// TwinCAT 3 PLC project CL_DefectManagerPLC
// Title: CL_DefectManager
// Company: CleanGreens SA
// Author: Massimo Lucano
// ProjectVersion: 2.4
// Description: class to handle defects. Majour upgrade with several fixes and dynamic allocation
// ProgramVersion: 3.1.4024.0
// libraries:
//   CL_ErrorsDatabase, * (CleanGreens SA)
//   CL_CleanGreensObjectsLibrary, * (CleanGreens SA)
//   Tc2_Database, * (Beckhoff Automation GmbH)
//   Tc2_DataExchange, * (Beckhoff Automation GmbH)
//   Tc2_Standard, * (Beckhoff Automation GmbH)
//   Tc2_System, * (Beckhoff Automation GmbH)
//   Tc2_Utilities, * (Beckhoff Automation GmbH)
//   Tc3_Database, * (Beckhoff Automation GmbH)
//   Tc3_Module, * (Beckhoff Automation GmbH)
// project tree:
//   DUTs/ E_DefectState.TcDUT, ST_DefectManagerConstants.TcDUT, ST_DefectTable.TcDUT, T_DefectErrorID.TcDUT (not stored), T_InstancePath.TcDUT
//   GVLs/ CDefect.TcGVL
//   / PlcTask.TcTTO
//   POUs/ CL_Defect.TcPOU, CL_DefectManager.TcPOU, ITF_Defect.TcIO

CONFIGURATION CL_DefectManagerPLC
    RESOURCE PLC ON TwinCAT3
        TASK PlcTask(INTERVAL := T#10ms, PRIORITY := 20);
        PROGRAM MAIN WITH PlcTask : MAIN;
    END_RESOURCE
END_CONFIGURATION

// ---- DUTs/E_DefectState.TcDUT
{attribute 'qualified_only' := ''}
//{attribute 'strict'}   without strict type casting between integer et enum types is possible
TYPE E_DefectState :
(
	None := 0,
	Off,
	Active,
	ActiveAndAck,
	OffAndNotAck
);
END_TYPE

// ---- DUTs/ST_DefectManagerConstants.TcDUT
TYPE ST_DefectManagerConstants :
STRUCT
  nMaxDefects	        : UINT;//maximun number of defects that can be registred in the defect manager
	nMaxDefectsView	    :	UINT;//number of line to show in the HMI, each line is a defect
  nNumIrrLinesForHMI  : UINT;//number of irrigation line handled by a single PLC and HMI
END_STRUCT
END_TYPE

// ---- DUTs/ST_DefectTable.TcDUT
TYPE ST_DefectTable :
STRUCT
  bHideDefect   : BOOL := TRUE;
  pDefect       : pointer to CL_Defect; //pointer to the Defect itself
	State         : E_DefectState := E_DefectState.None;
	Severity      : TcEventSeverity := TcEventSeverity.Verbose;
	ErrorID       : STRING(3) :='';
	ClassID       : STRING(3) :='';
	Color         : DWORD := 0;
  InstancePath  : T_InstancePath := '';
	Description   : T_MaxString := '';
	RisingEdge    : STRING(CDefect.nDefectTableStrLen_C) := '';;
	FallingEdge   : STRING(CDefect.nDefectTableStrLen_C) := '';;
END_STRUCT
END_TYPE

// ---- DUTs/T_InstancePath.TcDUT
TYPE T_InstancePath : STRING(512); END_TYPE

// ---- GVLs/CDefect.TcGVL
{attribute 'qualified_only'}
VAR_GLOBAL CONSTANT
  //Defect manager library constants max array size
  nDefectTableStrLen_C        : UINT := 40;
	nMaxDefects_C    		        : UINT := 1000;
	nMaxDefectsView_C           : UINT := 40;
  tInfoOffTimeout_C           : TIME := T#5S; 
  tInfoOffAndNotAckTimeout_C  : TIME := T#15S;
END_VAR

// ---- POUs/ITF_Defect.TcIO
INTERFACE ITF_Defect EXTENDS __SYSTEM.IQueryInterface

METHOD Ack
END_METHOD

METHOD PUBLIC BuildStringMsg : BOOL
//return false if no error 
VAR_INPUT
	sMsgOut_P   : POINTER TO T_StringBuffer;//return the Telegram message
  sTextOut_P  : POINTER TO T_StringBuffer;//return the ADS console message  
  stShow      : ST_ShowMsgFields;
END_VAR
END_METHOD

PROPERTY PUBLIC CanSendAlarmMsg : BOOL
GET
END_GET
END_PROPERTY

PROPERTY PUBLIC CanSendInfoMsg : BOOL
GET
END_GET
END_PROPERTY

PROPERTY PUBLIC CanSendRegisterMsg : BOOL
GET
END_GET
END_PROPERTY

PROPERTY ClassID : STRING(3)
GET
END_GET
END_PROPERTY

METHOD PUBLIC DefectSentToFalse
VAR_INPUT
END_VAR
END_METHOD

PROPERTY PUBLIC Description : String
GET
END_GET
END_PROPERTY

PROPERTY ErrorID : STRING(3)
GET
END_GET
END_PROPERTY

PROPERTY FallingEdge : DATE_AND_TIME
GET
END_GET
END_PROPERTY

PROPERTY PUBLIC HideDefect : bool
GET
END_GET
END_PROPERTY

PROPERTY InstancePath : T_InstancePath
GET
END_GET
END_PROPERTY

METHOD PUBLIC Register : BOOL
VAR_INPUT
	DefectMngr  : REFERENCE TO CL_DefectManager;
  inClassID	  :	STRING(3);
  inErrorID   :	STRING(3);
END_VAR
END_METHOD

PROPERTY RisingEdge : DATE_AND_TIME
GET
END_GET
END_PROPERTY

METHOD PUBLIC Set
VAR_INPUT
  bSetActivate : BOOL;
END_VAR
END_METHOD

METHOD PUBLIC SetOff
VAR_INPUT
END_VAR
END_METHOD

METHOD PUBLIC SetOn
VAR_INPUT
END_VAR
END_METHOD

METHOD PUBLIC SetOnWithMsg
VAR_INPUT
  sAddMsg_P     : POINTER TO T_MaxString;
END_VAR
END_METHOD

METHOD PUBLIC SetWithMsg
VAR_INPUT
  bSetActivate  : BOOL;
  sAddMsg_P     : POINTER TO T_MaxString;
END_VAR
END_METHOD

PROPERTY Severity : TcEventSeverity
GET
END_GET
END_PROPERTY

PROPERTY State : E_DefectState
GET
END_GET
END_PROPERTY

METHOD UpdateHideDefect
END_METHOD

END_INTERFACE

// ---- POUs/CL_Defect.TcPOU
{attribute 'reflection'}
FUNCTION_BLOCK CL_Defect IMPLEMENTS ITF_Defect
VAR
 	_State              : E_DefectState := E_DefectState.None; 
	
	_ErrorIndex					:	UDINT;
	_ClassIndex					:	UDINT;
	
  _ErrorID            : STRING(3);
  _ClassID            : STRING(3);
  
	_DefectMngr	        : REFERENCE TO CL_DefectManager;
	_bRegistered		    : BOOL := FALSE;
	
	_Severity           : TcEventSeverity := TcEventSeverity.Critical;//temporary solution without database
		
	//used to send Telegram msg
	bTelAlarmSent       : BOOL := FALSE;
  bTelInfoSent        : BOOL := FALSE;
	bTelRegisteredSent	: BOOL := FALSE;
  
  bHideDefect	        : BOOL := true;
	
	_RisingEdge         : DATE_AND_TIME;
	_FallingEdge		    : DATE_AND_TIME;
	
	{attribute 'instance-path'}
	{attribute 'no_init'}
	_InstancePath       : T_InstancePath;
	InstanceStr_P		    : POINTER TO T_StringBuffer;
  _sAddMsg		        : string(64) := '';
END_VAR

METHOD PUBLIC Ack
IF State = E_DefectState.Active THEN
  _State := E_DefectState.ActiveAndAck;
ELSIF State = E_DefectState.OffAndNotAck THEN
  _State := E_DefectState.Off;
	DefectSentToFalse();
END_IF
END_METHOD

METHOD PUBLIC BuildStringMsg : BOOL
//return false if no error 
VAR_INPUT
	sMsgOut_P       : POINTER TO T_StringBuffer;//return the Telegram message
  sTextOut_P      : POINTER TO T_StringBuffer;//return the ADS console message  
  stShow          : ST_ShowMsgFields;
END_VAR
VAR
	bTmpErr			    : BOOL;
	bTmp1Err		    : BOOL;
  nErrIdOut       : UDINT;
	fbFormatStr	    : FB_FormatString;
  
	severityStr	    : T_MaxString;
	stateStr        : T_MaxString;
	sMsgAddLine	    :	T_MaxString;
  sMsgTmp         : T_MaxString;
  sClassID        : T_MaxString;
  sErrorID        : T_MaxString;
END_VAR
BuildStringMsg := FALSE;
sClassID := _ClassID;
sErrorID := _ErrorID;

CASE _State OF
		E_DefectState.None : stateStr := 'None';
		E_DefectState.Off : stateStr := 'Off';
		E_DefectState.Active : stateStr := 'Active';
		E_DefectState.ActiveAndAck : stateStr := 'ActiveAndAck';
		E_DefectState.OffAndNotAck : stateStr := 'OffAndNotAck';
END_CASE

CASE _Severity OF
		TcEventSeverity.Critical : severityStr := 'Critical';
		TcEventSeverity.Error : severityStr := 'Error';
		TcEventSeverity.Info : severityStr := 'Info';
		TcEventSeverity.Verbose : severityStr := 'Verbose';
		TcEventSeverity.Warning : severityStr := 'Warning';
END_CASE

IF stShow.bTxtLog AND (sTextOut_P<>0) THEN 
  // Shorter, because issue for too long strings 
  IF _DefectMngr.NumIrrLinesForHMI <= 1 THEN
    IF _DefectMngr.MRCIrrLine = 0 THEN
      sMsgAddLine := UINT_TO_STRING(_DefectMngr.MRCIrrLineFixedID);
      sMsgAddLine := concat('Main cabinet ',sMsgAddLine);
      sMsgAddLine := concat(sMsgAddLine,' - ');
    ELSE
      sMsgAddLine := UINT_TO_STRING(_DefectMngr.MRCIrrLineFixedID);
      sMsgAddLine := concat('Line ',sMsgAddLine);
      sMsgAddLine := concat(sMsgAddLine,' - ');    
		END_IF
  ELSE
    IF _DefectMngr.MRCIrrLine = 0 THEN
      sMsgAddLine := 'for all lines';
      sMsgAddLine := concat('Main cabinet ',sMsgAddLine);
      sMsgAddLine := concat(sMsgAddLine,' - ');
    ELSE
      sMsgAddLine := UINT_TO_STRING(_DefectMngr.MRCIrrLine);
      sMsgAddLine := concat('Line ',sMsgAddLine);
      sMsgAddLine := concat(sMsgAddLine,' - ');
 	  END_IF
  END_IF
  
  fbFormatStr(
    sFormat	:= '$N Severity: %s  Status: %s  ClassID: %s  ErrID: %s $N InstancePath: %s $N Message sender: %s', 
    arg1  := F_STRING(severityStr),
    arg2	:= F_STRING(stateStr),
    arg3	:= F_STRING(sClassID),
    arg4	:= F_STRING(sErrorID), 
    arg5	:= F_STRING(_InstancePath),
    arg6  := F_STRING(sMsgAddLine),
    bError => bTmp1Err,  
    nErrId => nErrIdOut, 
    sOut	=> sTextOut_P^);
  
  IF bTmp1Err THEN
    sMsgTmp := ' FB_FormatStr Error : $N ';
    bTmp1Err := NOT CONCAT2(sTextOut_P,ADR(sMsgTmp),sTextOut_P,SIZEOF(T_StringBuffer));
    sMsgTmp := UDINT_TO_STRING(nErrIdOut);
    bTmp1Err := NOT CONCAT2(sTextOut_P,ADR(sMsgTmp),sTextOut_P,SIZEOF(T_StringBuffer));
    sMsgTmp := ' $N ';
    bTmp1Err := NOT CONCAT2(sTextOut_P,ADR(sMsgTmp),sTextOut_P,SIZEOF(T_StringBuffer));
	END_IF
 
  //concat class description short
  IF NOT bTmpErr THEN
    sMsgTmp := _DefectMngr.ErrorDB.GetClassShortMsg(_ClassIndex);
    sMsgTmp := concat(sMsgTmp,'$N');
    bTmpErr := NOT CONCAT2(sTextOut_P,ADR(sMsgTmp),sTextOut_P,SIZEOF(T_StringBuffer));
  END_IF	
   
  //concat error description short
  IF NOT bTmp1Err THEN
    sMsgTmp := ' Message description: ';	
    bTmp1Err := NOT CONCAT2(sTextOut_P,ADR(sMsgTmp),sTextOut_P,SIZEOF(T_StringBuffer));
  END_IF
  IF NOT bTmp1Err THEN
    sMsgTmp := _DefectMngr.ErrorDB.GetErrorShortMsg(_ErrorIndex);     
    bTmp1Err := NOT CONCAT2(sTextOut_P,ADR(sMsgTmp),sTextOut_P,SIZEOF(T_StringBuffer));
  END_IF	
  
  //add AddMsg string to the alarm message
  IF _sAddMsg <> '' THEN
    IF NOT bTmp1Err THEN
      sMsgTmp := '$N';	
      bTmp1Err := NOT CONCAT2(sTextOut_P,ADR(sMsgTmp),sTextOut_P,SIZEOF(T_StringBuffer));
    END_IF
    IF NOT bTmp1Err THEN
      bTmp1Err := NOT CONCAT2(sTextOut_P,ADR(_sAddMsg),sTextOut_P,SIZEOF(T_StringBuffer));
    END_IF	
	END_IF
  
  //concat twice new line
  IF NOT bTmp1Err THEN
    sMsgTmp := ' $N $N';	
    bTmp1Err := NOT CONCAT2(sTextOut_P,ADR(sMsgTmp),sTextOut_P,SIZEOF(T_StringBuffer));
  END_IF  
ELSE
  bTmp1Err := TRUE;
END_IF

//Telegram API new line character is %0A
//to insert it inside format string the Telegram use %%0A, while inside concat use %0A
//build the sMsgOut_P string buffers used to sent Telegram message
IF sMsgOut_P <>0 THEN
	bTmpErr := FALSE;
	IF stShow.bIstance THEN 
		fbFormatStr(
      sFormat	:= '%%0ASeverity: %S  Status: %S  ClassID: %S  ErrID: %S %%0AInstancePath: %S %%0AMessage sender: %s',
      arg1  := F_STRING(severityStr),
      arg2	:= F_STRING(stateStr),
      arg3	:= F_STRING(sClassID),
      arg4	:= F_STRING(sErrorID), 
      arg5	:= F_STRING(_InstancePath),
      arg6  := F_STRING(sMsgAddLine),    
      bError	=> bTmpErr,  
      nErrId	=> nErrIdOut, 
      sOut	=> sMsgOut_P^);
	ELSE
		fbFormatStr(
      sFormat	:= '%%0ASeverity: %S  Status: %S  ClassID: %S  ErrID: %S %%0AMessage sender: %s',
      arg1  := F_STRING(severityStr),
      arg2	:= F_STRING(stateStr),
      arg3	:= F_STRING(sClassID),
      arg4	:= F_STRING(sErrorID), 
      arg5  := F_STRING(sMsgAddLine),    
      bError	=> bTmpErr,  
      nErrId	=> nErrIdOut, 
      sOut	=> sMsgOut_P^);
	END_IF
  
  //build class description
  IF stShow.bLongClass THEN
    sMsgTmp := _DefectMngr.ErrorDB.GetClassLongMsg(_ClassIndex);
  ELSE
    sMsgTmp := _DefectMngr.ErrorDB.GetClassShortMsg(_ClassIndex);
	END_IF  
  IF NOT bTmpErr THEN
    sMsgTmp := concat(sMsgTmp,'%0A');
    bTmpErr := NOT CONCAT2(sMsgOut_P,ADR(sMsgTmp),sMsgOut_P,SIZEOF(T_StringBuffer));
  END_IF	
  
  //build error description either long or short
  IF NOT bTmpErr THEN
    sMsgTmp := 'Message description:%0A';	
    bTmpErr := NOT CONCAT2(sMsgOut_P,ADR(sMsgTmp),sMsgOut_P,SIZEOF(T_StringBuffer));
  END_IF
  IF stShow.bLongError THEN
    sMsgTmp := _DefectMngr.ErrorDB.GetErrorLongMsg(_ErrorIndex);
  ELSE
    sMsgTmp := _DefectMngr.ErrorDB.GetErrorShortMsg(_ErrorIndex);
	END_IF  
  IF NOT bTmpErr THEN
    bTmpErr := NOT CONCAT2(sMsgOut_P,ADR(sMsgTmp),sMsgOut_P,SIZEOF(T_StringBuffer));
  END_IF	
  
  IF _sAddMsg <> '' THEN
    IF NOT bTmp1Err THEN
      sMsgTmp := '%0A';	
      bTmp1Err := NOT CONCAT2(sMsgOut_P,ADR(sMsgTmp),sMsgOut_P,SIZEOF(T_StringBuffer));
    END_IF
    IF NOT bTmp1Err THEN
      bTmp1Err := NOT CONCAT2(sMsgOut_P,ADR(_sAddMsg),sMsgOut_P,SIZEOF(T_StringBuffer));
    END_IF	
	END_IF

  //build remed description
  IF NOT bTmpErr AND stShow.bRemed THEN
    sMsgAddLine := '%0A Correction:%0A';
    bTmpErr := NOT CONCAT2(sMsgOut_P,ADR(sMsgAddLine),sMsgOut_P,SIZEOF(T_StringBuffer));
  END_IF   
  IF NOT bTmpErr AND stShow.bRemed THEN
    sMsgTmp := _DefectMngr.ErrorDB.GetErrorRemedMsg(_ErrorIndex);
    bTmpErr := NOT CONCAT2(sMsgOut_P,ADR(sMsgTmp),sMsgOut_P,SIZEOF(T_StringBuffer));
  END_IF
  
END_IF//sMsgOut_P <>0 THEN
BuildStringMsg := NOT(bTmpErr OR bTmp1Err);
END_METHOD

PROPERTY PUBLIC CanSendAlarmMsg : BOOL
GET
CanSendAlarmMsg := NOT bTelAlarmSent AND _bRegistered;
if CanSendAlarmMsg then
  bTelAlarmSent := TRUE;
end_if
END_GET
END_PROPERTY

PROPERTY PUBLIC CanSendInfoMsg : BOOL
GET
CanSendInfoMsg := NOT bTelInfoSent AND _bRegistered;
if CanSendInfoMsg then
  bTelInfoSent := TRUE;
end_if
END_GET
END_PROPERTY

PROPERTY PUBLIC CanSendRegisterMsg : BOOL
GET
CanSendRegisterMsg := NOT bTelRegisteredSent AND _bRegistered;//bTelRegisteredSent = false only at Init time
if CanSendRegisterMsg then
  bTelRegisteredSent := TRUE;
end_if
END_GET
END_PROPERTY

PROPERTY PUBLIC ClassID : STRING(3)
GET
ClassID := _ClassID;
END_GET
END_PROPERTY

METHOD PUBLIC DefectSentToFalse
VAR_INPUT
END_VAR
bTelAlarmSent := FALSE;
bTelInfoSent := FALSE;
END_METHOD

PROPERTY PUBLIC DefectToSend : BOOL
GET
//condition OR pDf^.State = E_DefectState.OffAndNotAck added MPL date 16-11-2024
DefectToSend := State = E_DefectState.Active OR State = E_DefectState.ActiveAndAck OR State = E_DefectState.OffAndNotAck;
END_GET
END_PROPERTY

PROPERTY PUBLIC Description : String
GET
//Description := CONCAT(_ErrorLongMsg,_RemedMsg);
Description := _DefectMngr.ErrorDB.GetErrorShortMsg(_ErrorIndex);
END_GET
END_PROPERTY

PROPERTY PUBLIC ErrorID : STRING(3);
GET
ErrorID := _ErrorID;
END_GET
END_PROPERTY

PROPERTY PUBLIC FallingEdge : DATE_AND_TIME
GET
FallingEdge := _FallingEdge;
END_GET
END_PROPERTY

METHOD FB_init : BOOL
VAR_INPUT
	bInitRetains	: BOOL; // if TRUE, the retain variables are initialized (warm start / cold start)
	bInCopyCode		: BOOL;  // if TRUE, the instance afterwards gets moved into the copy code (online change)
END_VAR
VAR
	pos					  : UDINT;
END_VAR
InstanceStr_P := ADR(_InstancePath);
//BUG in FB_IotHttpRequest: cannot build the URL with the name of Project in it; why!! otherwise the URL 
//sent to Telegram Web API return server error.  Remove from the instance string the name of the project!
//find the first occurence of '.'
pos := FIND2(InstanceStr_P,ADR('.'));
DELETE2(InstanceStr_P,InstanceStr_P,SIZEOF(InstanceStr_P^),pos,1);//delete project name
//find the second occurence of '.'
pos := FIND2(InstanceStr_P,ADR('.'));
DELETE2(InstanceStr_P,InstanceStr_P,SIZEOF(InstanceStr_P^),pos,1);//delete PLC name
END_METHOD

PROPERTY PUBLIC HideDefect : bool
GET
HideDefect := bHideDefect;
END_GET
END_PROPERTY

PROPERTY PUBLIC InstancePath : T_InstancePath
GET
InstancePath := _InstancePath;
END_GET
END_PROPERTY

METHOD PUBLIC Register : BOOL
VAR_INPUT
	DefectMngr    : REFERENCE TO CL_DefectManager;
  inClassID	    :	STRING(3);
  inErrorID     :	STRING(3);
END_VAR
VAR
	i                   : UINT;
	ArrayIsFull         : INT;
	indDefectLine       : UDINT;
	DefectNumericStruct	:	ST_classAndErrorNum;
END_VAR
Register := _bRegistered := FALSE;
IF __ISVALIDREF(DefectMngr) THEN 
  _ErrorID := inErrorID;
  _ClassID := inClassID;
  
  bHideDefect := true;
	_DefectMngr REF= DefectMngr;
  
  //this part of code was not inside IF __ISVALIDREF(DefectManager)...we have to check before all that the reference to the DefectManager is good
  // Only way to have access to elements of an object stored into another one: method to extract the whole object!
  // TwinCAT or ST limitations!
  _DefectMngr.SearchDefectDB(errorID := inErrorID, classID := inClassID, udiDBErrorIndex => _ErrorIndex, udiDBClassIndex => _ClassIndex);
  
  (*
  DefectNumericStruct := _DefectMngr.ErrorDB.GetNumerics(udiErrorIndex := _ErrorIndex, udiClassIndex := _ClassIndex);  @@really buggy this method sometime it return ErrorID or ClassID wrong sometime not!!
  _ErrorID  := DefectNumericStruct.errorId; // Now, three digits IDs!
  _ClassID  := DefectNumericStruct.classId;	// Relation between classes and error IDs done in ST code again! (unique errorIDs across the classes)
  *)
  
  CASE _DefectMngr.ErrorDB.WhichSeverity(_ErrorIndex) OF
      0:  _Severity := TcEventSeverity.Verbose;
      1:  _Severity := TcEventSeverity.Info;
      2:  _Severity := TcEventSeverity.Warning;
      3:  _Severity := TcEventSeverity.Error;
      4:  _Severity := TcEventSeverity.Critical;
  END_CASE
	
	FOR i:= 1 TO _DefectMngr.nMaxDefects DO	
		IF (i = _DefectMngr.nMaxDefects) AND (_DefectMngr.ListAll(i,0) = 0) THEN // List of Defects is already full => Error
      _DefectMngr.ArrayIsFull := TRUE;
      ADSLOGSTR(ADSLOG_MSGTYPE_MSGBOX, 'Fatal error: too many defects: increase the array size and recompile','');
		ELSIF _DefectMngr.ListAll(i,0) = THIS THEN // Defect already in the list
      Register := _bRegistered := TRUE;
			EXIT;
		ELSIF _DefectMngr.ListAll(i,0) = 0 THEN // Add Defect in the list
			_DefectMngr.ListAll(i,THIS);
			Register := _bRegistered := TRUE;
			EXIT;
		END_IF
	END_FOR
  
END_IF
END_METHOD

PROPERTY PUBLIC RisingEdge : DATE_AND_TIME
GET
RisingEdge := _RisingEdge;
END_GET
END_PROPERTY

METHOD PUBLIC Set
VAR_INPUT
  bSetActivate : BOOL;
END_VAR
IF bSetActivate AND State <> E_DefectState.Active AND State <> E_DefectState.ActiveAndAck THEN
  _State := E_DefectState.Active;
  _RisingEdge	:= _DefectMngr._objActTime_R.GetDateTime;
  _FallingEdge := DT#1970-1-1-0:0:0;//DATE_AND_TIME#1970-1-1-0:0:0
  UpdateHideDefect();
ELSIF NOT bSetActivate THEN
	IF State = E_DefectState.Off OR State = E_DefectState.OffAndNotAck THEN
    //IMPORTANT: Alarm and Info messages can be sent again only if the Defect return to E_DefectState.Off
    IF State = E_DefectState.Off THEN
		  DefectSentToFalse();
    END_IF
	END_IF
  IF State = E_DefectState.Active THEN
    _State := E_DefectState.OffAndNotAck;
		_FallingEdge	:= _DefectMngr._objActTime_R.GetDateTime;//_DefectMngr.ActTime;
    UpdateHideDefect();
  ELSIF State = E_DefectState.ActiveAndAck THEN
    _State := E_DefectState.Off;
		_FallingEdge := _DefectMngr._objActTime_R.GetDateTime;//_DefectMngr.ActTime;
    UpdateHideDefect();
  ELSIF State = E_DefectState.None THEN
    _State := E_DefectState.Off;
    UpdateHideDefect();
	END_IF
END_IF
END_METHOD

METHOD PUBLIC SetOff
VAR_INPUT
END_VAR
Set(false);
END_METHOD

METHOD PUBLIC SetOn
VAR_INPUT
END_VAR
Set(TRUE);
END_METHOD

METHOD PUBLIC SetOnWithMsg
VAR_INPUT
    sAddMsg_P     : POINTER TO T_MaxString;
END_VAR
_sAddMsg := sAddMsg_P^;
Set(TRUE);
END_METHOD

METHOD PUBLIC SetWithMCErrorID
VAR_INPUT
  bSetActivate  : BOOL;
  MCErrorID     : UDINT;
END_VAR
_sAddMsg := UDINT_TO_STRING(MCErrorID);
_sAddMsg := concat(' MC Error ID : ',_sAddMsg);
Set(bSetActivate);
END_METHOD

METHOD PUBLIC SetWithMsg
VAR_INPUT
  bSetActivate  : BOOL;
  sAddMsg_P     : POINTER TO T_MaxString;
END_VAR
_sAddMsg := sAddMsg_P^;
Set(bSetActivate);
END_METHOD

PROPERTY Severity : TcEventSeverity
GET
Severity := _Severity;
END_GET
END_PROPERTY

PROPERTY State : E_DefectState
GET
State := _State;
END_GET
END_PROPERTY

METHOD UpdateHideDefect
bHideDefect := NOT (State = E_DefectState.Off) and NOT (State = E_DefectState.OffAndNotAck ) and not (State = E_DefectState.Active );
END_METHOD

END_FUNCTION_BLOCK

// ---- POUs/CL_DefectManager.TcPOU
{attribute 'enable_dynamic_creation'}
FUNCTION_BLOCK PUBLIC CL_DefectManager EXTENDS CL_MasterRootClass
VAR
	bInit			              : BOOL := FALSE;
	pDefect                 : POINTER TO CL_Defect;
	iDefect                 : ITF_Defect;
	stEmptyList             : ST_DefectTable;
	lTemp                   : BOOL;
	iShow                   : INT := 1;
  
  _WarningIsPresent       : BOOL;
  _ErrorIsPresent         : BOOL;
  _CriticalIsPresent      : BOOL;
  	
	// Constant values stored there (library ready)
	_nMaxDefectsView        :	UINT;
	_nMaxDefects            :	UINT;
  
  _nNumIrrLinesForHMI     : UINT;
  
  i1,x1,y1                : UINT;
  	
  AllDefects_ARP          : POINTER TO ARRAY[1..CDefect.nMaxDefects_C] OF POINTER TO CL_Defect; //used by CL_defect
  CurrentAllDefects_ARP   : POINTER TO ARRAY[1..CDefect.nMaxDefectsView_C] OF ST_DefectTable; // AllDefects_ARP^ of Defects activated 
  
  // Check by severity level
	DefaultAlarmIsPresent   : BOOL := FALSE;
	DefaultWarningIsPresent : BOOL := FALSE;

	bArrayIsFull            : BOOL := FALSE;

  //objects
	_objErrorDB_R	          :	REFERENCE TO CL_ErrorDB;
  _objActTime_R           :	REFERENCE TO CL_ActTimeDate;

  //-------------------------------------  HMI interface ---------------------------------------
  CurrentDefects_AR       : ARRAY[1..CDefect.nMaxDefectsView_C] OF ST_DefectTable; //For HMI, AllDefects_ARP^ of Defects shown
  CurrentDefectsInfo_AR   : ARRAY[1..CDefect.nMaxDefectsView_C] OF ST_DefectTable; //For HMI, AllDefects_ARP^ of Info Verbose Defects shown
  
  //HMI buttons interface
  Ack_Defects             : BOOL := FALSE;
  Ack_InfoVerboseDefects  : BOOL := FALSE;

  //button filter minimum level shown
	eMinSeverityShow        : TcEventSeverity  := TcEventSeverity.Info; 
  
	//button expert view; used only in HMI
	ExpertView              : BOOL := FALSE;

  // Color for HMI
	SeverityColor_Debug     : DWORD := 4294918837;
	SeverityColor_Info      : DWORD := 4278190335;
	SeverityColor_Warning   : DWORD := 4294945792;
	SeverityColor_Error     : DWORD := 4294901760;
	SeverityColor_Critical  : DWORD := 4288217088;
END_VAR

(*
Defect Critical -> Irrigation system state machine generates Abort, message generated is visible inside the Alarms HMI, send to Telegram operator group
Defect Error -> Irrigation system state machine generates Stop, message generated is visible inside the Alarms HMI, send to Telegram operator group
Defect Warning -> Irrigation system state machine generates no Stop or Abort, message generated is visible inside the Alarms HMI, send to Telegram operator group
IMPORTANT: warning defect can by promoted to Error after a while -> update ErrorDB
Defect Info -> Irrigation system state machine no Stop or Abort at all, only a message is generated visible inside the Infos HMI, send to Telegram operator group
Defect Verbose -> Irrigation system state machine So stop or Abort at all, only a message is generated visible to the Administrator Infos HMI, send to Telegram Debug group
TcEventSeverity : (Verbose:=0, Info:=1, Warning:=2, Error:=3, Critical:=4);
*)
IF bInit THEN
  THIS^.Run();
END_IF

PROPERTY PUBLIC ActTime : Reference to CL_ActTimeDate
GET
ActTime ref= _objActTime_R;
END_GET
END_PROPERTY

METHOD PUBLIC AllocateArrays : BOOL
VAR
  structSize			: UDINT;
	arraySize				: UDINT;
  i               : UINT;
END_VAR
//AllDefects_ARP array allocated in memory from 0..C.nMaxDefects_C
structSize := SIZEOF(CL_Defect);
arraySize := structSize * (_nMaxDefects+2);
AllDefects_ARP := __NEW(BYTE, arraySize);

structSize := SIZEOF(ST_DefectTable);
arraySize := structSize * (_nMaxDefectsView+2);
(*
CurrentDefects_ARP := __NEW(BYTE, arraySize);
CurrentDefectsInfo_ARP := __NEW(BYTE, arraySize);	
*)
arraySize := structSize * (_nMaxDefectsView+2);//*2
CurrentAllDefects_ARP := __NEW(BYTE, arraySize);

(*
AllocateArrays :=  AllDefects_ARP <> 0 AND CurrentDefects_ARP <> 0 AND 
                  CurrentDefectsInfo_ARP <> 0 AND 
                  CurrentAllDefects_ARP <> 0;
*)
AllocateArrays :=  AllDefects_ARP <> 0 AND  CurrentAllDefects_ARP <> 0;

IF AllocateArrays THEN 
  FOR i := 1 TO _nMaxDefects DO
    AllDefects_ARP^[i] := 0; //At init, set all Defects pointer to 0
  END_FOR
  FOR i := 1 TO _nMaxDefectsView DO
    CurrentAllDefects_ARP^[i].InstancePath     := '';
    CurrentAllDefects_ARP^[i].bHideDefect      := TRUE;
    CurrentAllDefects_ARP^[i].State            := E_DefectState.None;
    CurrentAllDefects_ARP^[i].Severity         := TcEventSeverity.Verbose;
    CurrentAllDefects_ARP^[i].ErrorID          := '';
    CurrentAllDefects_ARP^[i].ClassID          := '';
    CurrentAllDefects_ARP^[i].Description      := '';
    CurrentAllDefects_ARP^[i].RisingEdge       := '';
    CurrentAllDefects_ARP^[i].FallingEdge      := '';
    CurrentAllDefects_ARP^[i].Color := 0;
  
    CurrentDefects_AR[i] := stEmptyList;    
    CurrentDefectsInfo_AR[i] := stEmptyList;
  END_FOR
END_IF
END_METHOD

PROPERTY AreCriticalDefects : bool
GET
AreCriticalDefects := _CriticalIsPresent;
END_GET
SET // PUBLIC
_CriticalIsPresent := AreCriticalDefects;
END_SET
END_PROPERTY

PROPERTY AreErrorDefects : bool
GET
AreErrorDefects := _ErrorIsPresent;
END_GET
SET // PUBLIC
_ErrorIsPresent := AreErrorDefects;
END_SET
END_PROPERTY

PROPERTY AreWarningDefecsts : bool
GET
AreWarningDefecsts := _WarningIsPresent;
END_GET
SET // PUBLIC
_WarningIsPresent := AreWarningDefecsts;
END_SET
END_PROPERTY

PROPERTY PUBLIC ArrayIsFull : BOOL
GET
ArrayIsFull := bArrayIsFull;
END_GET
SET // PUBLIC
bArrayIsFull := ArrayIsFull;
END_SET
END_PROPERTY

PROPERTY PUBLIC ErrorDB : reference TO CL_ErrorDB
GET
//objErrorDB := ADR(_objErrorDB);
ErrorDB REF= _objErrorDB_R;
END_GET
END_PROPERTY

METHOD PUBLIC Init : BOOL
VAR_INPUT
  stIrrLine           : ST_LineReference;
  ErrorDB_R           : REFERENCE TO CL_ErrorDB;
  ActTime_R           : REFERENCE TO CL_ActTimeDate;
  stDefectManager_C   : ST_DefectManagerConstants;
END_VAR
bInit := Init := FALSE;
IF NOT bInit AND __ISVALIDREF(ErrorDB_R) AND __ISVALIDREF(ActTime_R) AND 
 stDefectManager_C.nMaxDefects > 0 AND stDefectManager_C.nMaxDefects <= CDefect.nMaxDefects_C 
 AND stDefectManager_C.nMaxDefectsView > 0 AND stDefectManager_C.nMaxDefectsView <= CDefect.nMaxDefectsView_C AND stDefectManager_C.nNumIrrLinesForHMI > 0 THEN
  
  MRCLineRef := stIrrLine;
  _nMaxDefects	:=	stDefectManager_C.nMaxDefects;
  _nMaxDefectsView	:=	stDefectManager_C.nMaxDefectsView;
  _nNumIrrLinesForHMI := stDefectManager_C.nNumIrrLinesForHMI;

  _objErrorDB_R REF= ErrorDB_R;
  _objActTime_R REF= ActTime_R;
  
  IF AllDefects_ARP = 0 AND CurrentAllDefects_ARP = 0 THEN
    //Arrays not already allocated
    bInit := Init := AllocateArrays();
  ELSE
    //Arrays already allocated
    bInit := Init := TRUE;
  END_IF
END_IF
END_METHOD

METHOD PUBLIC ListAll : POINTER TO CL_Defect
VAR_INPUT
	ind     : UINT;
	defect  : POINTER TO CL_Defect;
END_VAR
IF (ind > 0) AND (ind <= _nMaxDefects) AND AllDefects_ARP <> 0 THEN 
	IF defect <> 0 THEN 
		AllDefects_ARP^[ind] := defect;
		ListAll := defect;
	ELSE
		ListAll := AllDefects_ARP^[ind];
		defect := AllDefects_ARP^[ind];
	END_IF
END_IF
END_METHOD

METHOD PUBLIC ListCurrent : POINTER TO CL_Defect
VAR_INPUT
	ind     : UINT;
END_VAR
VAR
  pDf : pointer to CL_Defect;
END_VAR
ListCurrent := 0;
IF (ind > 0) AND (ind <= _nMaxDefectsView) THEN 
  IF Len2(ADR(CurrentAllDefects_ARP^[ind].InstancePath)) > 0 THEN
    pDf := CurrentAllDefects_ARP^[ind].pDefect;
	  ListCurrent := CurrentAllDefects_ARP^[ind].pDefect;
  END_IF
END_IF
END_METHOD

PROPERTY PUBLIC nMaxDefects : UINT
GET
nMaxDefects	:=	_nMaxDefects;
END_GET
END_PROPERTY

PROPERTY PUBLIC nMaxDefectsView : UINT
GET
nMaxDefectsView	:= _nMaxDefectsView;
END_GET
END_PROPERTY

PROPERTY PUBLIC NumIrrLinesForHMI : UINT
GET
NumIrrLinesForHMI := _nNumIrrLinesForHMI;
END_GET
END_PROPERTY

METHOD PUBLIC Release : BOOL
VAR_INPUT
END_VAR
bInit := FALSE;
IF AllDefects_ARP <> 0  THEN 
  __DELETE(AllDefects_ARP);
END_IF

(*
IF CurrentDefects_ARP <> 0 THEN 
  //__DELETE(CurrentDefects_ARP);
END_IF
IF CurrentDefectsInfo_ARP <> 0 THEN 
  __DELETE(CurrentDefectsInfo_ARP);
END_IF
IF CurrentDefectsVerbose_ARP <> 0 THEN 
  __DELETE(CurrentDefectsVerbose_ARP);
END_IF
*)

IF CurrentAllDefects_ARP <> 0 THEN 
  __DELETE(CurrentAllDefects_ARP);
END_IF

//Release := AllDefects_ARP = 0 AND CurrentDefects_ARP = 0 AND CurrentDefectsInfo_ARP = 0 AND CurrentDefectsVerbose_ARP = 0 AND CurrentAllDefects_ARP = 0;
Release := AllDefects_ARP = 0 AND CurrentAllDefects_ARP = 0;
END_METHOD

METHOD PRIVATE Run
(*
Defect Critical -> Irrigation system state machine generates Abort, message generated is visible inside the Alarms HMI, send to Telegram operator group
Defect Error -> Irrigation system state machine generates Stop, message generated is visible inside the Alarms HMI, send to Telegram operator group
Defect Warning -> Irrigation system state machine generates no Stop or Abort, message generated is visible inside the Alarms HMI, send to Telegram operator group
IMPORTANT: warning defect can by promoted to Error after a while -> update ErrorDB
Defect Info -> Irrigation system state machine no Stop or Abort at all, only a message is generated visible inside the Infos HMI, send to Telegram operator group
Defect Verbose -> Irrigation system state machine So stop or Abort at all, only a message is generated visible to the Administrator Infos HMI, send to Telegram Debug group
TcEventSeverity : (Verbose:=0, Info:=1, Warning:=2, Error:=3, Critical:=4);
Critical, Error, Warning are found if state is: E_DefectState.Active OR E_DefectState.ActiveAndAck OR E_DefectState.OffAndNotAck
//MPL 16-11-2024 added condition "OR State = E_DefectState.OffAndNotAck" -> the error or critical or warning is found even if Off but not Ack 
*)
iShow := 1;
//at each PLC cycle the Run method is executed and so the DefectManager check again if a Critical, Error, Warning defect is present
_CriticalIsPresent := FALSE;
_ErrorIsPresent := FALSE;
_WarningIsPresent := FALSE;
FOR i1:= 1 TO _nMaxDefects DO // C.nNbrMaxDefects_C DO
  IF AllDefects_ARP^[i1] <> 0 THEN // Check if one Defect is registred at this index
    iDefect := AllDefects_ARP^[i1]^;
    IF __QUERYPOINTER(iDefect, pDefect) THEN // Ctrl if address has the good interface (ITF_Defect)
      Run_HandleAckByVISU();
      
      IF pDefect^.State = E_DefectState.Off OR pDefect^.State = E_DefectState.None THEN
        Run_RemoveAllDefectsOffOrNone();
      ELSIF pDefect^.State = E_DefectState.Active OR pDefect^.State = E_DefectState.ActiveAndAck OR pDefect^.State = E_DefectState.OffAndNotAck THEN
        //MPL 16-11-2024 added condition OR pDefect^.State = E_DefectState.OffAndNotAck -> the error or critical or warning is found even if Off but not Ack
        Run_AddAllDefectsPresent();
        Run_AutoOffInfoVerbose();
        Run_FindAllCriticalErrorWarning();
      END_IF
      
      (*IF pDefect^.State = E_DefectState.Active OR pDefect^.State = E_DefectState.ActiveAndAck OR pDefect^.State = E_DefectState.OffAndNotAck THEN
        //find all Active defects 
        Run_FindAllCriticalErrorWarning();
      END_IF*)
      
    END_IF//IF __QUERYPOINTER(iDefect, pDefect)
	END_IF//IF AllDefects_ARP^[i1] <> 0
END_FOR

FOR y1:= 1 TO _nMaxDefectsView DO //C.nMaxDefectsView_C DO
  CurrentDefects_AR[y1] := stEmptyList;
  CurrentDefectsInfo_AR[y1] := stEmptyList;
END_FOR

//TcEventSeverity : (Verbose:=0, Info:=1, Warning:=2, Error:=3, Critical:=4);
IF eMinSeverityShow < TcEventSeverity.Warning  THEN 
  //only Warning:=2, Error:=3, Critical:=4 are transferred
  eMinSeverityShow := TcEventSeverity.Warning;
END_IF

FOR i1:= 1 TO _nMaxDefectsView DO// Why a double for loop here? Maybe a better way.
  //TcEventSeverity : (Verbose:=0, Info:=1, Warning:=2, Error:=3, Critical:=4);
  
  //eMinSeverityShow >= Warning, thus verbose and info are not transferred in CurrentDefects_AR
  IF  CurrentAllDefects_ARP^[i1].Severity >= eMinSeverityShow THEN
    FOR y1:= 1 TO _nMaxDefectsView DO //C.nMaxDefectsView_C DO
      IF CurrentDefects_AR[y1].InstancePath = '' THEN
        CurrentDefects_AR[y1] := CurrentAllDefects_ARP^[i1];
        EXIT;
			END_IF
		END_FOR
	END_IF
  
  //only Info = 1 and Verbose = 0 are transferred in CurrentDefectsInfo_AR
  IF  CurrentAllDefects_ARP^[i1].Severity <= TcEventSeverity.Info THEN
    FOR y1:= 1 TO _nMaxDefectsView DO //C.nMaxDefectsView_C DO
      IF CurrentDefectsInfo_AR[y1].InstancePath = '' THEN
        CurrentDefectsInfo_AR[y1] := CurrentAllDefects_ARP^[i1];
        EXIT;
			END_IF
		END_FOR
	END_IF

END_FOR
END_METHOD

METHOD PRIVATE Run_AddAllDefectsPresent
// Add in the AllDefects_ARP^ all defects present
lTemp := FALSE;
FOR y1:= 1 TO _nMaxDefectsView DO
  IF CurrentAllDefects_ARP^[y1].InstancePath = pDefect^.InstancePath THEN
    //CurrentAllDefects_ARP^[y1].pDefect := pDefect;
    CurrentAllDefects_ARP^[y1].State := pDefect^.State;
    SetEdgeStr(pDefect^.RisingEdge, CurrentAllDefects_ARP^[y1].RisingEdge);
    SetEdgeStr(pDefect^.FallingEdge, CurrentAllDefects_ARP^[y1].FallingEdge);
    lTemp := TRUE;
    iShow := iShow + 1;
    EXIT;
  END_IF
END_FOR
IF NOT lTemp THEN
  FOR y1:= 1 TO _nMaxDefectsView DO
    IF CurrentAllDefects_ARP^[y1].InstancePath = '' THEN
      CurrentAllDefects_ARP^[y1].pDefect := pDefect;
      CurrentAllDefects_ARP^[y1].InstancePath     := pDefect^.InstancePath;
      CurrentAllDefects_ARP^[y1].bHideDefect      := pDefect^.HideDefect;
      CurrentAllDefects_ARP^[y1].State            := pDefect^.State;
      CurrentAllDefects_ARP^[y1].Severity         := pDefect^.Severity;
      CurrentAllDefects_ARP^[y1].ErrorID          := pDefect^.ErrorID;
      CurrentAllDefects_ARP^[y1].ClassID          := pDefect^.ClassID;
      CurrentAllDefects_ARP^[y1].Description      := pDefect^.Description;
      SetEdgeStr(pDefect^.RisingEdge, CurrentAllDefects_ARP^[y1].RisingEdge);
      SetEdgeStr(pDefect^.FallingEdge, CurrentAllDefects_ARP^[y1].FallingEdge);
      CASE pDefect^.Severity OF
        TcEventSeverity.Verbose   : CurrentAllDefects_ARP^[y1].Color := SeverityColor_Debug;
        TcEventSeverity.Info      : CurrentAllDefects_ARP^[y1].Color := SeverityColor_Info;
        TcEventSeverity.Warning   : CurrentAllDefects_ARP^[y1].Color := SeverityColor_Warning;
        TcEventSeverity.Error     : CurrentAllDefects_ARP^[y1].Color := SeverityColor_Error;
        TcEventSeverity.Critical  : CurrentAllDefects_ARP^[y1].Color := SeverityColor_Critical;
      END_CASE
      iShow := iShow + 1;
      EXIT;
    END_IF
  END_FOR
END_IF
END_METHOD

METHOD PRIVATE Run_AutoOffInfoVerbose
VAR
  lifeTime : TIME;
  //dt1,dt2 :  DATE_AND_TIME;
END_VAR
//TcEventSeverity : (Verbose:=0, Info:=1, Warning:=2, Error:=3, Critical:=4);        
IF  pDefect^.Severity <= TcEventSeverity.Info THEN
  //dt1 := ActTime.GetDateTime;
  //dt2 := pDefect^.RisingEdge;
  lifeTime := ActTime.GetDateTime - pDefect^.RisingEdge;
  IF lifeTime >= CDefect.tInfoOffAndNotAckTimeout_C AND pDefect^.State <> E_DefectState.OffAndNotAck THEN //execute only once  C.tInfoOffAndNotAckTimeout_C := T#30S;
    //automatically set Defect to Off and NotAck
    pDefect^.Set(FALSE);
  END_IF
  lifeTime := ActTime.GetDateTime - pDefect^.FallingEdge;
  IF lifeTime >= CDefect.tInfoOffTimeout_C THEN
    IF pDefect^.State = E_DefectState.OffAndNotAck THEN //execute only once   C.tInfoOffTimeout_C := T#10S; 
      //automatically set Defect to Off
      pDefect^.Ack();
    END_IF
  ELSE
    if pDefect^.State <> E_DefectState.Active and pDefect^.State <> E_DefectState.OffAndNotAck then
      pDefect^.DefectSentToFalse();
    end_if
  END_IF
END_IF
END_METHOD

METHOD PRIVATE Run_FindAllCriticalErrorWarning
IF pDefect^.Severity = TcEventSeverity.Critical THEN
  _CriticalIsPresent := TRUE;
END_IF
IF pDefect^.Severity = TcEventSeverity.Error THEN
  _ErrorIsPresent  := TRUE;
END_IF
IF pDefect^.Severity = TcEventSeverity.Warning THEN
  _WarningIsPresent := TRUE;
END_IF
END_METHOD

METHOD private Run_HandleAckByVISU
//TcEventSeverity : (Verbose:=0, Info:=1, Warning:=2, Error:=3, Critical:=4);   
//Ack Info and Verbose     
IF  pDefect^.Severity <= TcEventSeverity.Info AND Ack_InfoVerboseDefects THEN
  pDefect^.Ack();
END_IF

//Ack Warning:=2, Error:=3, Critical:=4
IF pDefect^.Severity > TcEventSeverity.Info AND Ack_Defects THEN
  pDefect^.Ack();
END_IF
END_METHOD

METHOD PRIVATE Run_RemoveAllDefectsOffOrNone
//Remove all defects from AllDefects_ARP^ Defect with state off or none
FOR y1 := 1 TO _nMaxDefectsView DO //C.nMaxDefectsView_C DO
  IF CurrentAllDefects_ARP^[y1].InstancePath = pDefect^.InstancePath THEN
      CurrentAllDefects_ARP^[y1] := stEmptyList;
      // Move UP all alarms in the AllDefects_ARP^
      FOR x1 := y1 TO _nMaxDefectsView-1 DO//??? _nMaxDefectsView-1
        CurrentAllDefects_ARP^[x1] := CurrentAllDefects_ARP^[x1+1];
      END_FOR
  END_IF
END_FOR
END_METHOD

METHOD PUBLIC SearchDefectDB
VAR_INPUT
  errorID	:	STRING(3);
	classID	:	STRING(3);
END_VAR
VAR_OUTPUT
//	errorValues:	ST_SP_RecordReturn;
//	classValues:	ST_SP_ClassReturn;
	udiDBErrorIndex	:	UDINT;
	udiDBClassIndex	:	UDINT;
  error:  BOOL;
END_VAR
VAR
	bExecEnd:		BOOL;
	uiSafeIter:	USINT := 0;
END_VAR
_objErrorDB_R.SearchErrorData(errorID := errorID, udiErrorIndex => udiDBErrorIndex, error => error);
_objErrorDB_R.SearchClassData(classID := classID, udiClassIndex => udiDBClassIndex, error => error);
END_METHOD

METHOD PRIVATE SetEdgeStr
VAR_INPUT
  dtEdge : DATE_AND_TIME;
END_VAR
VAR_IN_OUT
  sEdge  : STRING(CDefect.nDefectTableStrLen_C);
END_VAR
VAR
  sMonth  : T_MaxString;
  sDay    : T_MaxString;
  sTmp    : T_MaxString;
END_VAR
IF dtEdge > DT#1970-1-1-0:0:0 AND sEdge = '' THEN
  sTmp := DT_TO_STRING(dtEdge);
  sTmp := DELETE(sTmp, 8, 1); //DELETE(sTmp, 6, 0); 
  sTmp := REPLACE(sTmp, ' ',1,6);
  sMonth := Left(sTmp,2);
  sTmp := DELETE(sTmp, 4, 0); 
  sDay := Left(sTmp,2);
  sTmp := DELETE(sTmp, 3, 0);
  sDay := concat(sDay,'/');
  sDay := concat(sDay, sMonth);
  sTmp := concat(sDay,sTmp);
  sEdge := sTmp;
END_IF
END_METHOD

METHOD private SevereDefectSet : BOOL
VAR
	i			: UINT;	
	pDef	: POINTER TO CL_Defect;
	iDef	: ITF_Defect;
END_VAR
// this funtion return true if AT LEAST one defect critical or warning or error is set
SevereDefectSet := FALSE;
FOR i:= 1 TO _nMaxDefects DO
	IF AllDefects_ARP^[i] <> 0 THEN // Check if one defect is registred at this index
		iDef := AllDefects_ARP^[i]^;
		// Ctrl if address has the good interface (ITF_Default)
		IF __QUERYPOINTER(iDef, pDef) THEN 
			IF pDef^.State = E_DefectState.Active OR pDef^.State = E_DefectState.OffAndNotAck OR pDef^.State = E_DefectState.ActiveAndAck THEN
				IF pDef^.Severity = TcEventSeverity.Critical OR pDef^.Severity = TcEventSeverity.Error OR pDef^.Severity = TcEventSeverity.Warning THEN
					SevereDefectSet := TRUE;
					EXIT;
				END_IF
			END_IF
		END_IF
	END_IF
END_FOR
END_METHOD

END_FUNCTION_BLOCK
